{attribute 'qualified_only'}
VAR_GLOBAL CONSTANT
	SUCCESS		: Strings.Str := 'Success';
	FAIL		: Strings.Str := 'Fail';
	SAME		: Strings.Str := 'Same';
END_VAR

(* stored: Version 1.1.0.1
   GVL CState: Id {fcc3794d-0502-4b10-a5b1-1fb168391c12} *)
